RoboDK station: Large Table with corner axis.rdk

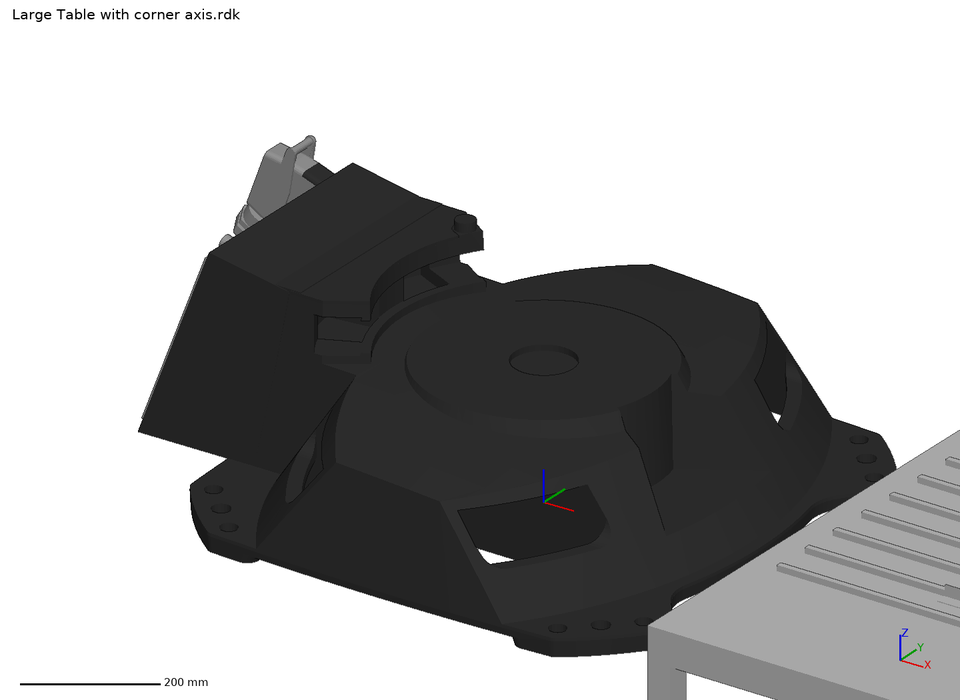
[picture v0: the station drawn from its stored meshes, robots at their saved joint values, targets as dots, program paths as lines]
Station Large Table with corner axis (saved by RoboDK 5.2.3). Poses are relative to the parent item; angles as X-Y-Z fixed-axis rotations.
  - frame KUKA KR 210 R2700 extra Base at (0, 0, 0) mm
    - robot KUKA KR 210 R2700 extra: 6 axes, payload 210 kg, reach 2696 mm, repeatability 0.06 mm, weight 1068 kg
        joint limits [-185, -140, -120, -350, -125, -350] to [185, -5, 155, 350, 125, 350]; home [0, -90, 90, 0, 0, 0]; saved at [32.784, -5.411, 22.473, 211.742, 116.949, 68.427]
      - tool Spindle, TCP at (278.6, 0, 88) mm, rotated rx 0 ry 90 rz 0 deg, size 85 x 346.5 x 128 mm
  - frame Corner First Plate at (2495, 660, 510.8) mm, rotated rx 0 ry 0 rz 90 deg
  - object Table 3 at (1700, -800, 455) mm, rotated rx 0 ry 0 rz 90 deg, size 1820 x 1600 x 475 mm, geometry from Table 3.stl
